// TwinCAT 3 PLC project PLC1
// ProgramVersion: 3.1.4024.0
// libraries:
//   Tc2_Standard, * (Beckhoff Automation GmbH)
//   Tc2_System, * (Beckhoff Automation GmbH)
//   Tc3_Module, * (Beckhoff Automation GmbH)
// project tree:
//   GVLs/ DB2_Counters.TcGVL, DIDO.TcGVL
//   / PlcTask.TcTTO
//   POUs/ FB2_Counters.TcPOU, MAIN.TcPOU
// real-time tasks:
//   TASK PlcTask: cycle T#10ms, priority 20, ADS port 350
// I/O:
//   DEVICE Device 1 (EtherCAT), AmsNetId 10.10.10.3.2.1
//     Term 1 (EK1100) [EK1100 EtherCAT Coupler (2A E-Bus)]
//       Term 2 (EL2004) [EL2004 4Ch. Dig. Output 24V, 0.5A]
// variable links:
//   PLC1/PLC1 Instance <-> Device 1 (EtherCAT)/Term 1 (EK1100)/Term 2 (EL2004)
//     PlcTask Outputs/DIDO.Uitgang{1..4} <-> Channel {1..4}/Output  (4 links)

CONFIGURATION PLC1
    RESOURCE PLC ON TwinCAT3
        TASK PlcTask(INTERVAL := T#10ms, PRIORITY := 20);
        PROGRAM MAIN WITH PlcTask : MAIN;
    END_RESOURCE
END_CONFIGURATION

// ---- GVLs/DB2_Counters.TcGVL
{attribute 'qualified_only'}
VAR_GLOBAL
	eenHzTrigger : BOOL;
END_VAR

// ---- GVLs/DIDO.TcGVL
{attribute 'qualified_only'}
VAR_GLOBAL
	
	 
	Uitgang1 AT %QX26.0 : BOOL := FALSE;
	Uitgang2 AT %QX26.1 : BOOL := FALSE;
	Uitgang3 AT %QX26.2 : BOOL := FALSE;
	Uitgang4 AT %QX26.3 : BOOL := FALSE;
	
END_VAR

// ---- POUs/MAIN.TcPOU
PROGRAM MAIN
VAR
    toggleOutput : BOOL := FALSE; // Output toggles every 5 seconds
    timer        : TON;           // Timer function block
    timerPeriod  : TIME := T#5s;  // Duration for high and low states
END_VAR


// Timer logic
timer.IN := TRUE;            // Timer always runs
timer.PT := timerPeriod;     // Set the timer duration

// Toggle logic
IF timer.Q THEN
    toggleOutput := NOT toggleOutput; // Toggle the output
    timer(IN := FALSE);               // Reset the timer
    timer(IN := TRUE);                // Restart the timer
END_IF

// Call the timer block
timer();
DIDO.Uitgang1 := toggleOutput;

END_PROGRAM

// ---- POUs/FB2_Counters.TcPOU
FUNCTION_BLOCK FB2_Counters
VAR_INPUT
	ENable: Bool;
END_VAR
VAR_OUTPUT
END_VAR
VAR
END_VAR

VAR_STAT
	eenHzTrig: R_TRIG := FALSE;
END_VAR

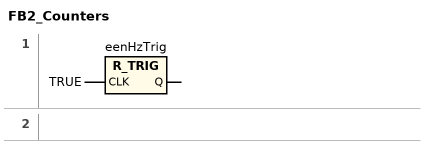
// NETWORK 1
eenHzTrig(CLK := TRUE); // R_TRIG

// NETWORK 2

END_FUNCTION_BLOCK
